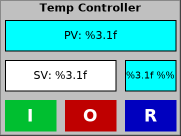
VISUALIZATION VFM_TempController  // 181x136
VAR_IN_OUT
	HMI: ST_HMI_TempController;
END_VAR
    Rectangle (0,0 181x136), "Temp Controller"
    Rectangle (5,20 171x31), "PV: %3.1f", text variable: HMI.Status.Actual, input disabled if: NOT HMI.Status.Enabled
    Rectangle (5,60 111x31), "SV: %3.1f", text variable: HMI.Config.Param.Setpoint, input disabled if: NOT HMI.Status.Enabled
        OnMouseClick: write the text variable via Default
    Rectangle (5,100 51x31), "I", input disabled if: NOT HMI.Command.Manual
        tap HMI.Command.Start
    Rectangle (125,100 51x31), "R", input disabled if: NOT HMI.Command.Manual
        tap HMI.Command.ResetPID
    Rectangle (65,100 51x31), "O", input disabled if: NOT HMI.Command.Manual
        tap HMI.Command.Stop
    Rectangle (125,60 51x31), "%3.1f %%", text variable: HMI.Status.CtrlOutput, input disabled if: NOT HMI.Status.Enabled
END_VISUALIZATION

(* stored: Version 1.1.0.1, ProductVersion 3.1.4024.12
   Visu VFM_TempController: Id {13cd0614-274d-4e7b-8ef7-bf33f543102e} *)
